TYPE "sCTRL_SUP_CSS"
TITLE =User data type for CTRL-SUP-CSS Codac States
AUTHOR  : ITER
FAMILY  : SDD

	STRUCT
		VAR1 : BYTE ;						 // VAR1
	END_STRUCT ;
END_TYPE

//----------------------------------------------------------------------------------


DATA_BLOCK "CodacStates"
TITLE =Data block for Codac States
AUTHOR  : ITER
FAMILY  : SDD

	STRUCT
	Header : "CodacStatesHeader" ;
	CTRL_SUP_CSS : "sCTRL_SUP_CSS" ;		// CS-Studio tools test
   Footer : "CodacStatesFooter" ;
  END_STRUCT ;
BEGIN
   Header.Length := 64;		// Length of "CodacStates" DB
   Header.InterfaceVersion := '01-19-2016 09:37:09' ;
END_DATA_BLOCK



DATA_BLOCK "CodacChannels"
TITLE =Data block for Codac communication parameters
AUTHOR  : ITER
FAMILY  : SPSS

  STRUCT
   channel1 : "UCodacChannel" ;	//State and configuration
   channel2 : "UCodacChannel" ;	//Simple commands
  END_STRUCT ;
BEGIN
   channel1.SEND_LEN := 64;		// Length of "CodacStates" DB
   channel1.RECV_LEN := 0 ;		// Length of "CodacConfiguration" DB
   channel2.SEND_LEN := 0 ;
   channel2.RECV_LEN := 0 ;		// Length of "CodacCommands" DB
END_DATA_BLOCK


